Staubli VAL3: insert_aCOunt.pgx

public program insert_aCount(string x_sItem (dimensions=1), bool x_bActive (dimensions=1), aio x_aDio (dimensions=1))
begin
  // insert a new IO
  if isDefined(aCount[x_sItem])==false and ioStatus(x_aDio)>=0
    insert(aCount[x_sItem])
    aCount[x_sItem].bActive=x_bActive
    aCount[x_sItem].sID=x_sItem
    aCount[x_sItem].sName=x_sItem
    aioLink(aCount[x_sItem].aAio,x_aDio)
    aCount[x_sItem].bEnable=true
  endIf
end
